TYPE "AreaConfig"
VERSION : 0.1
// Block: AreaConfig
   STRUCT
      TimeOutStopImmediate : Time;
      TimeOutStopInPhase : Time;
      TimeOutStopProgrammed : Time;
      TimeOutResetAlarms : Time;
   END_STRUCT;

END_TYPE
